TYPE Room_State_DemandHeating_Hmi :
STRUCT
END_STRUCT
END_TYPE

(* stored: Version 1.1.0.1
   DUT Room_State_DemandHeating_Hmi: Id {20902f1a-b815-4cae-b018-4d258d23364b} *)
